TYPE EtcMasterBase_62654B43 :
STRUCT
END_STRUCT
END_TYPE

(* stored: Version 1.2.0.0, ProductVersion 3.1.4024.11
   DUT EtcMasterBase_62654B43: Id {89bdb7d4-60b1-42d8-b563-25f1dfdb776d} *)
